// TIA Portal V16 export
// export: Created 2024-12-03T15:41:39.4768861Z, ExportSetting WithDefaults, DisplayName Totally Integrated Automation Portal, DisplayVersion V16 Update 6, DisplayName TIA Portal Version Control Interface, DisplayVersion V16 Update 2, DisplayName TIA Portal Openness, DisplayVersion V16 Update 6, DisplayName TIA Portal Teamcenter Gateway, DisplayVersion V16, DisplayName SINAMICS Startdrive Advanced, DisplayVersion V16 Update 5, DisplayName SINAMICS Startdrive G130, G150, S120, S150, SINAMICS MV, S210, DisplayVersion V16 Update 5, DisplayName SINAMICS Startdrive G110M, G120, G120C, G120D, G120P, G115D, DisplayVersion V16 Update 5, DisplayName STEP 7 Professional, DisplayVersion V16 Update 6, DisplayName STEP 7 Safety, DisplayVersion V16, DisplayName WinCC Advanced / Unified PC, DisplayVersion V16 Update 6
FUNCTION_BLOCK "LightTowerController"   // FB58, SCL
{ S7_Optimized_Access := 'FALSE' }
VERSION : 0.1
// stored: AutoNumber true, IsIECCheckEnabled false, SetENOAutomatically false, UDAEnableTagReadback false
   VAR
      AutoModeOn : "SmartBool";
   END_VAR
   VAR DB_SPECIFIC
      StartupBuzzer : TOF_TIME;
   END_VAR
   VAR
      grav_226 : "LightTowerGravController";
      grav_227 : "LightTowerGravController";
      grav_236 { S7_SetPoint := 'True'} : "LightTowerGravController";
      grav_237 { S7_SetPoint := 'True'} : "LightTowerGravController";
      grav_256 { S7_SetPoint := 'True'} : "LightTowerGravController";
      grav_257 { S7_SetPoint := 'True'} : "LightTowerGravController";
      grav_266 { S7_SetPoint := 'True'} : "LightTowerGravController";
      grav_267 { S7_SetPoint := 'True'} : "LightTowerGravController";
      grav_276 { S7_SetPoint := 'True'} : "LightTowerGravController";
      grav_277 { S7_SetPoint := 'True'} : "LightTowerGravController";
      grav_286 { S7_SetPoint := 'True'} : "LightTowerGravController";
      grav_287 { S7_SetPoint := 'True'} : "LightTowerGravController";
      grav_519 { S7_SetPoint := 'True'} : "LightTowerGravController";
      grav_527 { S7_SetPoint := 'True'} : "LightTowerGravController";
      grav_528 { S7_SetPoint := 'True'} : "LightTowerGravController";
      grav_534 { S7_SetPoint := 'True'} : "LightTowerGravController";
   END_VAR
   VAR_TEMP
      T_Index : Int;
      T_StartLED : Bool;
      T_ResetLED : Bool;
   END_VAR
BEGIN
   REGION GLOBAL LIGHT TOWER SIGNALS

       REGION GREEN LED

           "Q_LED_GREEN" := 0;

           IF "ApplicationState_DB".Appstate[1].States.AutoModeActivated.State THEN
               "Q_LED_GREEN" := 1;
           END_IF;

       END_REGION

       REGION ORANGE LED

           "Q_LED_ORANGE" :=
           "ApplicationState_DB".GlobalState.States.AlarmActive AND "Clock_0.5Hz";

       END_REGION

       REGION RED LED

           "Q_LED_RED" :=
           NOT "ApplicationState_DB".Appstate[1].States.EmergencyOk.State;

       END_REGION

   END_REGION
END_FUNCTION_BLOCK
